// TIA Portal V20 export
// export: Created 2026-09-14T11:29:00.9812641Z, ExportSetting None, DisplayName Totally Integrated Automation Portal, DisplayVersion V20, DisplayName TIA Portal Openness, DisplayVersion V20, DisplayName TIA Portal Version Control Interface, DisplayVersion V20, DisplayName STEP 7 Professional, DisplayVersion V20, DisplayName STEP 7 Safety, DisplayVersion V20, DisplayName WinCC Basic/Comfort/Advanced, DisplayVersion V20, DisplayName WinCC Unified, DisplayVersion V20
TYPE "LMQTT_typeParamData"
   STRUCT
      connectFlag { S7_SetPoint := 'True'} : "LMQTT_typeConnectFlags";
      keepAlive : UInt := 30;   // KeepAlive in Seconds. 0=No Keepalive
      clientIdentifier : String[23] := 'Siemens SIMATIC';   // Unique name of the client used from the client to identify itself at the broker during the connection establishment
      willTopic : String[100];   // If the will flag is set, the topic for the last will need to be defined
      willMessage : String[100];   // If the will flag is set, the message for the last will needs to be defined
      userName : String[100];   // If the username flag is set, the username for the login at the broker needs to be defined
      password : String[200];   // If the password flag is set, the password for the login at the broker needs to be defined
   END_STRUCT;
END_TYPE
